FUNCTION_BLOCK FB_Stopper
VAR
	bStopperCylinder		AT%Q*		: BOOL; //Cylinder moves stopper down
	bStopperSensor			AT%I*		: BOOL; //Sensor checks if stopper is occupied
END_VAR

METHOD MoveStopper : BOOL
VAR
	Stopper:FB_Stopper;
END_VAR
IF NOT Stopper.Occupied THEN			//If stopper is nor occupied
	Stopper.StopperCylinder:=TRUE;		//Move stopper up
END_IF
END_METHOD

PROPERTY Occupied : BOOL
GET
Occupied:=bStopperSensor;
END_GET
END_PROPERTY

PROPERTY StopperCylinder : BOOL
SET
bStopperCylinder:=StopperCylinder;
END_SET
END_PROPERTY

METHOD StopperDown : BOOL
VAR
	Stopper:FB_Stopper;
END_VAR
IF NOT Stopper.Occupied THEN			//If stopper is nor occupied
	Stopper.StopperCylinder:=FALSE;		//Move stopper up
END_IF
END_METHOD

END_FUNCTION_BLOCK

(* stored: Version 1.1.0.1, ProductVersion 3.1.4024.12
   POU FB_Stopper: Id {383cb24f-2c1b-461f-b125-d95395c56095}, SpecialFunc None
   Method MoveStopper: Id {700460a4-e30d-4180-a344-992e4150cd33}
   Property Occupied: Id {604a1840-cb70-441d-ac6c-c026757b33ab}
   Get Get: Id {1e2eaaa3-99f3-4ba1-a8dc-81358aabc0ac}
   Property StopperCylinder: Id {a8613c54-93a1-498d-8726-3638d396650b}
   Set Set: Id {fc328863-6a3c-43df-baae-74e1926005bf}
   Method StopperDown: Id {78a327d4-05c4-470f-88ca-e4ddeb5918a0} *)
